PROGRAM getFlowrate
VAR

	flowrate: LREAL;
	poids_old: REAL;

END_VAR



VAR

END_VAR



flowrate := (Weight_Station1-poids_old)/20*3600/1000.0/1000.0;

poids_old := Weight_Station1;




flowrate := (Weight_Station2-poids_old)/20*3600/1000.0/1000.0;

poids_old := Weight_Station2;




flowrate := (Weight_Station3-poids_old)/20*3600/1000.0/1000.0;

poids_old := Weight_Station3;





flowrate := (Weight_Station4-poids_old)/20*3600/1000.0/1000.0;

poids_old := Weight_Station4;

END_PROGRAM

(* stored: Version 1.1.0.1, ProductVersion 3.1.0.26
   POU getFlowrate: Id {08292630-e839-4887-b390-a45ee2fcf8a3} *)
